Fanuc KAREL source: kt00004.compact.KL

PROGRAM KT00004
%STACKSIZE=65535
%PRIORITY=65535
%NOLOCKGROUP
VAR
I1 : INTEGER
R2 : REAL
OUT : REAL
BEGIN
I1=2
R2=3.0
OUT=((I1) + R2)
END KT00004
